// TIA Portal V17 export
// export: Created 2023-02-14T02:49:14.6209368Z, ExportSetting WithDefaults, DisplayName Totally Integrated Automation Portal, DisplayVersion V17, DisplayName TIA Portal Openness, DisplayVersion V17, DisplayName TIA Portal Teamcenter Gateway, DisplayVersion V17, DisplayName TIA Portal Version Control Interface, DisplayVersion V17, DisplayName SINAMICS Startdrive Advanced, DisplayVersion V17, DisplayName SINAMICS Startdrive G130, G150, S120, S150, SINAMICS MV, S210, DisplayVersion V17, DisplayName SINAMICS Startdrive G110M, G120, G120C, G120D, G120P, G115D, DisplayVersion V17, DisplayName STEP 7 Professional, DisplayVersion V17, DisplayName STEP 7 Safety, DisplayVersion V17, DisplayName WinCC Professional, DisplayVersion V17
DATA_BLOCK "MB to Osa"   // DB265
{ S7_Optimized_Access := 'FALSE' }
VERSION : 0.1
// stored: AutoNumber false, DBAccessibleFromOPCUA true, DBAccessibleFromWebserver true, IsOnlyStoredInLoadMemory false, IsWriteProtectedInAS false
   VAR
      HeartBeat : Bool;   // Clock 1Hz
      ChiliFresh1_Prod_Req : Bool;
      ChiliFresh2_Prod_Req : Bool;
      ChiliFresh3_Prod_Req : Bool;
      ChiliFresh1_Line_OK : Bool;
      ChiliFresh2_Line_OK : Bool;
      ChiliFresh3_Line_OK : Bool;
      ChiliFresh1_CIP_Enable : Bool;
      ChiliFresh2_CIP_Enable : Bool;
      ChiliFresh3_CIP_Enable : Bool;
      freeBool11 : Bool;
      freeBool12 : Bool;
      freeBool13 : Bool;
      freeBool14 : Bool;
      freeBool15 : Bool;
      freeBool16 : Bool;
      freeBool17 : Bool;
   END_VAR
BEGIN
END_DATA_BLOCK
